{attribute 'GeneratedUsingTerminal: EL9930-0001-0016'}
{attribute addProperty BoxType "EL9930-0001-0016"}
{attribute addProperty Id "IO_InputsEMPTY_STRUCTURE0IO_OutputsEMPTY_STRUCTURE0WcStateAT %I*WcState_9091E0EB2InfoDataAT %I*InfoData_6F19DB2B2"}
{attribute addProperty CRC "133970461"}
{attribute addProperty Size "4"}
TYPE EL9930_07FC3A1D :
STRUCT
	{attribute addProperty Name "IO_Inputs"}
	IO_Inputs : EMPTY_STRUCTURE;
	{attribute addProperty Name "IO_Outputs"}
	IO_Outputs : EMPTY_STRUCTURE;
	{attribute addProperty Name "WcState"}
	WcState : WcState_9091E0EB;
	{attribute addProperty Name "InfoData"}
	InfoData : InfoData_6F19DB2B;
END_STRUCT
END_TYPE

(* stored: Version 1.2.0.0, ProductVersion 3.1.4024.9
   DUT EL9930_07FC3A1D: Id {5de14868-224e-4e47-a9eb-7494cc48cf07} *)
